INTERFACE I_StateManager EXTENDS Debug.I_Debug

PROPERTY Current : Tags.I_Tag
GET
END_GET
END_PROPERTY

METHOD Get : Results.Result
VAR_INPUT
	nPos				: UDINT;
END_VAR
VAR_OUTPUT
	iTag				: Tags.I_Tag;
END_VAR
END_METHOD

METHOD GetOnChange : Broadcast.I_Signal
VAR_INPUT
END_VAR
END_METHOD

PROPERTY Pretender : Tags.I_Tag
GET
END_GET
END_PROPERTY

PROPERTY Previous : Tags.I_Tag
GET
END_GET
END_PROPERTY

METHOD Request : Results.Result
VAR_INPUT
	iTag		: Tags.I_Tag;
END_VAR
END_METHOD

END_INTERFACE

(* stored: Version 1.1.0.1
   Itf I_StateManager: Id {67b23057-fe11-433c-9a95-8419d40ab691}
   Folder Get: Id {9c864531-7425-40a4-b921-2fc1424e61d3}
   Folder Other: Id {955dd895-0d9a-4720-9ffb-e1afc4e3e76b}
   Folder Request: Id {776ea33a-e4cc-4e85-80e7-570bf87d0f8d}
   Folder State: Id {a33e3b7e-257a-4dcc-a64c-44af723e8245}
   Property Current: Id {8f090f85-2d74-4f4d-a840-95ecca29e2e1}
   Get Get: Id {01a1fb79-a945-4882-b795-3fa9280bb658}
   Method Get: Id {00765a51-51ae-4a3a-b27e-2c6218cca014}
   Method GetOnChange: Id {edb4bbce-eaa3-4c8b-990e-5b73f470f6c4}
   Property Pretender: Id {454bf289-44ab-4cab-ba74-955c038db8d1}
   Get Get: Id {e5bb54f5-c287-4267-af62-d366666ce4bd}
   Property Previous: Id {f52f561f-9cd2-48e3-b486-4cd0cfcc879a}
   Get Get: Id {7314605f-c57d-43ac-8f8c-2fb0fcd29f32}
   Method Request: Id {93e47a5c-1aaa-4a03-892c-23942c4e7ff6} *)
